TYPE ST_MoverConfig EXTENDS ST_MoveOnTrackOptions:
STRUCT
//Velocity (mm/s)
	MaxVelo			: LREAL := 4000;
	NormalVelo		: LREAL := 3800;
	StoppingVelo	: LREAL := 300;
//Acceleration (mm/s^2)
	NormalAccel		: LREAL := 4000;
	MaxAccel		: LREAL := 8000;
//Deceleration (mm/s^2)
	NormalDecel		: LREAL := 3000;	
	MaxDecel		: LREAL := 8000;
//Jerk (mm/s^3)
	NormalJerk		: LREAL := 10000;
	MaxJerk			: LREAL := 20000;
//Platooning Vars
	VeloComp		: LREAL := 600;
	NormalMoverGap	: LREAL := 800;
	TightMoverGap	: LREAL := 300;
END_STRUCT
END_TYPE

(* stored: Version 1.1.0.1
   DUT ST_MoverConfig: Id {b2784631-d9fa-04c5-02b3-42fadcc04d80} *)
